TYPE "Limits"
VERSION : 0.1
   STRUCT
      Min : "Val";
      Max : "Val";
   END_STRUCT;

END_TYPE

